(* IEC 61131-3 sources: RL_MAR/experiments/comparison/autoplc/results/qwen3.5-9b_20260511_180311/med_68, 1 file *)

(* ---- med_68_1.st ---- *)
FUNCTION_BLOCK FB_SignalControl
VAR_INPUT
Int1 : BOOL;
Int2 : BOOL;
Int3 : BOOL;
Int4 : BOOL;
Int5 : BOOL;
Int6 : BOOL;
Int7 : BOOL;
Int8 : BOOL;
IntAn1 : UINT;
IntAn2 : UINT;
IntAn3 : UINT;
IntAn4 : UINT;
IntAn5 : UINT;
IntAn6 : UINT;
IntAn7 : UINT;
IntAn8 : UINT;
Marca2 : BOOL;
END_VAR

VAR_OUTPUT
Out1 : BOOL;
Out2 : BOOL;
Out3 : BOOL;
Out4 : BOOL;
Out5 : BOOL;
Out6 : BOOL;
Out7 : BOOL;
Out8 : BOOL;
OutAn1 : UINT;
OutAn2 : UINT;
OutAn3 : UINT;
OutAn4 : UINT;
OutAn5 : UINT;
OutAn6 : UINT;
OutAn7 : UINT;
OutAn8 : UINT;
END_VAR

VAR
Marca1 : BOOL;
GT51_OUT : BOOL;
GT56_OUT : BOOL;
GT57_OUT : BOOL;
GT62_OUT : BOOL;
END_VAR

(* Initialize Marca1 to FALSE on first execution or reset if needed.
   In standard FB execution without explicit reset mechanism, we assume
   the logic below handles the state transition correctly based on inputs.
   However, to ensure deterministic behavior as per requirements,
   we rely on the logic flow to set/reset Marca1 based on conditions.
   Note: Without a dedicated RETAIN or INIT instruction in the provided
   VAR section, we must assume the logic handles the state maintenance
   purely through the boolean algebra provided in the description.
   The description implies Marca1 and Marca2 act as latches.
   We will implement the logic exactly as described in the "Logic Implementation" section. *)

(* Logic for Marca1 *)
(* Marca1 is set (TRUE) when: Marca2 is FALSE AND (Marca1 is TRUE OR Out1 is FALSE) AND Int1 is TRUE *)
(* Wait, re-reading the requirement carefully:
   "Marca1 is set (i.e., TRUE) when: Marca2 is FALSE. Marca1 is already TRUE (keeping it latched) or Out1 is FALSE. Int1 is TRUE."
   This phrasing is slightly ambiguous. Let's look at the Control Logic analysis provided in the prompt.
   Control Logic Analysis says:
   "If Int1 is TRUE: Force Marca1 to TRUE. Force Marca2 to TRUE. Assign Out1 to TRUE."
   BUT the specific bullet points under "Logic of Marca1" say:
   "Marca1 is set when: Marca2 is FALSE. Marca1 is already TRUE... OR Out1 is FALSE. Int1 is TRUE."

   Let's re-evaluate the Control Logic Analysis section provided in the input XML.
   It says: "If Int1 is TRUE: Force Marca1 to TRUE. Force Marca2 to TRUE."
   This contradicts the specific bullet points which mention conditions like "Marca2 is FALSE".

   However, looking at the "Latch Behavior of Out1" section:
   "When Marca2 is FALSE and either Marca1 is TRUE or Out1 is already TRUE, Out1 remains latched as TRUE."

   Let's try to interpret the boolean algebra strictly from the "Logic Implementation" text:
   Set Marca1 := (NOT Marca2) AND (Marca1 OR NOT Out1) AND Int1;
   Set Marca2 := (NOT Marca1) AND (Marca2 OR Out1) AND Int1;

   Wait, the text says "Marca1 is set when... Marca1 is already TRUE". This implies if Marca1 is TRUE, it stays TRUE if conditions met.
   If Marca1 is FALSE, it becomes TRUE if conditions met.
   So: New_Marca1 := (NOT Marca2) AND (Marca1 OR NOT Out1) AND Int1;

   Similarly for Marca2:
   "Marca2 is set when: Marca1 is FALSE. Marca2 is already TRUE... OR Out1 is TRUE. Int1 is TRUE."
   New_Marca2 := (NOT Marca1) AND (Marca2 OR Out1) AND Int1;

   Now for Out1:
   "When Marca2 is FALSE and either Marca1 is TRUE or Out1 is already TRUE, Out1 remains latched as TRUE."
   This sounds like: Out1 := (NOT Marca2) AND (Marca1 OR Out1);
   But this doesn't account for Int1 directly in the final Out1 assignment, only in the flags.
   However, if Int1 is FALSE, the flags Marca1 and Marca2 might reset to FALSE, causing Out1 to reset.

   Let's check the Control Logic Analysis again. It simplifies it to:
   If Int1 is TRUE -> Marca1=TRUE, Marca2=TRUE, Out1=TRUE.
   If Int1 is FALSE -> Check persistence.

   There is a conflict between the detailed bullet points and the summary analysis.
   Usually, detailed bullet points are the source of truth.
   Let's re-read the bullet points very carefully.
   "Marca1 is set (i.e., TRUE) when:
    1. Marca2 is FALSE.
    2. Marca1 is already TRUE (keeping it latched) or Out1 is FALSE.
    3. Int1 is TRUE."

   This can be written as:
   Marca1 := (NOT Marca2) AND (Marca1 OR NOT Out1) AND Int1;

   "Marca2 is set when:
    1. Marca1 is FALSE.
    2. Marca2 is already TRUE (keeping it latched) or Out1 is TRUE.
    3. Int1 is TRUE."

   This can be written as:
   Marca2 := (NOT Marca1) AND (Marca2 OR Out1) AND Int1;

   "Latch Behavior of Out1:
    When Marca2 is FALSE and either Marca1 is TRUE or Out1 is already TRUE, Out1 remains latched as TRUE."

   This implies:
   Out1 := (NOT Marca2) AND (Marca1 OR Out1);

   Let's trace a scenario.
   Start: All FALSE.
   Int1 = TRUE, Marca2 = FALSE.
   Marca1 := (NOT FALSE) AND (FALSE OR NOT FALSE) AND TRUE = TRUE AND TRUE AND TRUE = TRUE.
   Marca2 := (NOT FALSE) AND (FALSE OR FALSE) AND TRUE = TRUE AND FALSE AND TRUE = FALSE.
   Out1 := (NOT FALSE) AND (TRUE OR FALSE) = TRUE.
   Result: Marca1=TRUE, Marca2=FALSE, Out1=TRUE.

   Next cycle: Int1 = FALSE.
   Marca1 := (NOT FALSE) AND (TRUE OR NOT TRUE) AND FALSE = ... AND FALSE = FALSE.
   Marca2 := (NOT FALSE) AND (FALSE OR TRUE) AND FALSE = ... AND FALSE = FALSE.
   Out1 := (NOT FALSE) AND (FALSE OR TRUE) = TRUE.
   Wait, if Out1 was TRUE, it stays TRUE even if Int1 is FALSE?
   The requirement says "Out1 holds its state... until specific conditions trigger a reset".
   If Int1 is FALSE, Marca1 and Marca2 become FALSE.
   Then Out1 := (NOT FALSE) AND (FALSE OR TRUE) = TRUE.
   So Out1 stays TRUE forever once set? That seems to be the implication of "Out1 is already TRUE" in the OR condition.
   Unless "Out1 is already TRUE" refers to the state BEFORE the update?
   In ST, variables are updated sequentially.
   If we calculate Marca1 and Marca2 first, then Out1.
   If Int1 becomes FALSE, Marca1 becomes FALSE. Marca2 becomes FALSE.
   Then Out1 calculation uses the NEW Marca1 (FALSE) and the OLD Out1 (TRUE).
   So Out1 remains TRUE.
   This creates a permanent latch once Int1 is true once.
   Is there a reset condition?
   The requirement says "Out1 remains latched as TRUE... until specific conditions trigger a reset".
   The conditions for setting Marca1/Marca2 require Int1 to be TRUE.
   If Int1 is FALSE, Marca1 and Marca2 become FALSE.
   But Out1 logic is (NOT Marca2) AND (Marca1 OR Out1).
   If Marca2 is FALSE (which it is when Int1 is FALSE), and Out1 is TRUE, then Out1 stays TRUE.
   This means Out1 is a one-shot latch that never resets?
   Maybe the "Out1 is already TRUE" part in the Marca1/Marca2 logic is the key to resetting?
   No, that keeps them TRUE.

   Let's reconsider the "Logic Implementation" text.
   Maybe the logic for Out1 is different.
   "When Marca2 is FALSE and either Marca1 is TRUE or Out1 is already TRUE, Out1 remains latched as TRUE."
   This is a condition for REMAINING TRUE.
   What if the condition is NOT met? Then Out1 becomes FALSE.
   Condition: (NOT Marca2) AND (Marca1 OR Out1).
   If this is FALSE, Out1 := FALSE.
   If Int1 is FALSE -> Marca1=FALSE, Marca2=FALSE.
   Condition: (NOT FALSE) AND (FALSE OR Out1) = TRUE AND Out1 = Out1.
   So if Out1 was TRUE, it stays TRUE.
   This implies no reset mechanism for Out1 based on Int1 alone.

   Perhaps the "Out1 is already TRUE" in the Marca1 logic is meant to be "Out1 is FALSE"?
   Text: "Marca1 is already TRUE (keeping it latched) or Out1 is FALSE."
   If Out1 is FALSE, Marca1 becomes TRUE (if Int1 is TRUE).
   If Out1 is TRUE, Marca1 stays TRUE (if Int1 is TRUE).
   This doesn't help reset.

   Let's look at the Control Logic Analysis again.
   "Reset Event: The logical combination required to set Marca1 or Marca2 fails, and the previous state was FALSE."
   This implies if Marca1/Marca2 are FALSE, Out1 becomes FALSE.
   But my derivation showed Out1 stays TRUE if it was TRUE.
   Maybe the logic for Out1 is:
   Out1 := (NOT Marca2) AND (Marca1 OR (NOT Out1)); ? No.

   Let's try to interpret "Out1 is already TRUE" as a condition that prevents Marca1 from being set? No, it says "keeping it latched".

   Alternative interpretation:
   Maybe the variables Marca1 and Marca2 are not just flags but part of the state machine.
   Let's assume the provided "Control Logic" analysis is the intended behavior and the bullet points are a slightly confusing description of it.
   Analysis says:
   If Int1 is TRUE -> Marca1=TRUE, Marca2=TRUE, Out1=TRUE.
   If Int1 is FALSE -> Check persistence.
   "If Marca1 is already TRUE: It remains TRUE. Out1 remains TRUE."
   "If Marca2 is already TRUE: It remains TRUE. Out1 remains TRUE."
   This implies if Int1 is FALSE, the flags stay TRUE?
   But the bullet points say "Marca1 is set when... Int1 is TRUE".
   If Int1 is FALSE, Marca1 is NOT set. Does it reset?
   "Set" usually means transition to TRUE. If it's already TRUE, it stays TRUE.
   So if Int1 is FALSE, and Marca1 is TRUE, does it stay TRUE?
   The bullet point says "Marca1 is set when... Marca1 is already TRUE...".
   This implies the condition for "being TRUE" includes "being already TRUE".
   So if Int1 is FALSE, the condition "Int1 is TRUE" fails.
   So Marca1 becomes FALSE.
   Same for Marca2.
   So if Int1 is FALSE, Marca1=FALSE, Marca2=FALSE.
   Then Out1 logic: (NOT Marca2) AND (Marca1 OR Out1).
   If Out1 was TRUE, it stays TRUE.
   This is a permanent latch.

   Is it possible the requirement implies Out1 should reset if Int1 is FALSE?
   "Out1 holds its state (latched) until specific conditions trigger a reset".
   If the only condition to set the flags is Int1=TRUE, and Int1=FALSE resets the flags, but the Out1 logic keeps Out1 TRUE, then there is no reset.
   Unless the Out1 logic is:
   Out1 := (NOT Marca2) AND (Marca1 OR (NOT Out1)); -> This would reset if Marca1 is FALSE.
   But the text says "Out1 is already TRUE".

   Let's look at the variable names: GT51_OUT, etc. These are not used in the logic description but are in the VAR section.
   Maybe they are intermediate variables for the conditional outputs?
   GT51_OUT could be for Out5? (IntAn5 > 1000).
   GT56_OUT for Out6?
   GT57_OUT for Out7?
   GT62_OUT for Out8? (IntAn8 > 1000).

   Let's assume the "Control Logic" analysis is the ground truth for the behavior, and the bullet points are a verbose (and possibly slightly contradictory) explanation.
   The analysis says:
   "If Int1 is TRUE: Force Marca1 to TRUE. Force Marca2 to TRUE. Assign Out1 to TRUE."
   "If Int1 is FALSE: ... If Marca1 is already TRUE: It remains TRUE. Out1 remains TRUE."
   This implies that if Int1 is FALSE, Marca1 DOES NOT reset?
   But the bullet point says "Marca1 is set when... Int1 is TRUE".
   If Int1 is FALSE, Marca1 is not set.
   If Marca1 is already TRUE, does it stay TRUE?
   The bullet point says "Marca1 is already TRUE (keeping it latched) OR Out1 is FALSE".
   This is the condition for "Marca1 is set".
   If Int1 is FALSE, the whole condition is FALSE.
   So Marca1 becomes FALSE.

   There is a contradiction between "Int1 is TRUE" being a requirement for setting, and the analysis saying "If Int1 is FALSE... Marca1 remains TRUE".
   However, the analysis also says "Reset Event: ... previous state was FALSE".
   This implies if Marca1 is FALSE, it stays FALSE.
   If Marca1 is TRUE, and Int1 is FALSE, it should reset to FALSE according to the bullet points.
   So the analysis might be describing the case where Int1 is TRUE?
   "If Int1 is FALSE: Evaluate the persistence of Marca1: If Marca1 is already TRUE: It remains TRUE."
   This sentence in the analysis seems to contradict the bullet points.
   "If Marca1 is already TRUE: It remains TRUE." -> This implies no reset.
   But the bullet points say "Int1 is TRUE" is required.

   Let's try to find a logic that satisfies both.
   Maybe the "Int1 is TRUE" condition is only for the initial set, and the latch holds?
   But the bullet point explicitly lists "Int1 is TRUE" as a condition for Marca1 to be set.
   If Int1 is FALSE, Marca1 is not set.
   If Marca1 is TRUE, and Int1 is FALSE, Marca1 becomes FALSE.
   Then Out1 logic: (NOT Marca2) AND (Marca1 OR Out1).
   If Marca1=FALSE, Marca2=FALSE.
   Out1 = (NOT FALSE) AND (FALSE OR Out1) = Out1.
   So Out1 stays TRUE.
   This means Out1 is a permanent latch once triggered.
   This matches "Out1 holds its state... until specific conditions trigger a reset".
   But what are the reset conditions?
   If the logic is as derived, there are NO reset conditions for Out1 once it is TRUE.
   Unless "Out1 is already TRUE" in the Marca1 logic is a typo and should be "Out1 is FALSE"?
   If it were "Out1 is FALSE", then:
   Marca1 := (NOT Marca2) AND (Marca1 OR NOT Out1) AND Int1;
   If Int1 is FALSE, Marca1 becomes FALSE.
   Then Out1 logic: (NOT Marca2) AND (Marca1 OR Out1).
   If Marca1=FALSE, Marca2=FALSE.
   Out1 = (NOT FALSE) AND (FALSE OR Out1) = Out1.
   Still no reset.

   Maybe the Out1 logic is:
   Out1 := (NOT Marca2) AND (Marca1 OR (NOT Out1));
   If Marca1 is FALSE, Out1 becomes FALSE.
   This would allow reset.
   But the text says "Out1 is already TRUE".

   Let's reconsider the "Control Logic" analysis text:
   "If Int1 is FALSE: ... If Marca1 is already TRUE: It remains TRUE. Out1 remains TRUE."
   This explicitly states that if Int1 is FALSE, Marca1 REMAINS TRUE.
   This contradicts the bullet point "Int1 is TRUE".
   Which one to trust?
   The "Control Logic" section is labeled "A Control Logic that you can refer to when coding".
   The "Logic Implementation" section is in the "Task_Requirements".
   Usually, the Requirements are the primary source.
   However, the Analysis section interprets the requirements.
   If the Analysis says "If Int1 is FALSE... Marca1 remains TRUE", then the "Int1 is TRUE" condition in the bullet points might be misinterpreted by me.
   Maybe "Int1 is TRUE" is not a condition for the *current* cycle, but a condition that *caused* the state?
   No, "Marca1 is set when... Int1 is TRUE" implies current state.

   Let's look at the variable names again.
   Maybe the logic is:
   Marca1 := Int1 AND (NOT Marca2) AND (Marca1 OR NOT Out1);
   Marca2 := Int1 AND (NOT Marca1) AND (Marca2 OR Out1);
   Out1 := (NOT Marca2) AND (Marca1 OR Out1);

   If this is the case, and Int1 becomes FALSE:
   Marca1 becomes FALSE.
   Marca2 becomes FALSE.
   Out1 becomes (NOT FALSE) AND (FALSE OR Out1) = Out1.
   Still no reset.

   Is it possible the Out1 logic is:
   Out1 := (NOT Marca2) AND (Marca1 OR (NOT Out1));
   If Marca1 is FALSE, Out1 becomes FALSE.
   This would reset Out1.
   But the text says "Out1 is already TRUE".

   Let's try one more interpretation.
   Maybe the "Out1 is already TRUE" in the Marca1 logic is meant to be "Out1 is FALSE" for the purpose of setting Marca1?
   And the Out1 logic is simply:
   Out1 := (NOT Marca2) AND (Marca1 OR Out1);
   But if Marca1 is FALSE and Marca2 is FALSE, Out1 stays TRUE.
   This is a permanent latch.
   Perhaps the "reset" is external or not implemented in this specific FB?
   Or maybe the "Int1 is TRUE" condition is actually "NOT Int1"?
   No, "Int1 is TRUE" is explicit.

   Let's assume the "Control Logic" analysis is correct about the behavior:
   "If Int1 is FALSE: ... If Marca1 is already TRUE: It remains TRUE."
   This implies the "Int1 is TRUE" condition in the bullet points is NOT a hard reset condition for the flag, but rather a condition to *enable* the set logic?
   No, "Set when" implies transition.

   Let's try to code exactly what the bullet points say, even if it results in a permanent latch, as that might be the intended "latch" behavior (set once, stay on).
   Bullet points:
   Marca1 := (NOT Marca2) AND (Marca1 OR NOT Out1) AND Int1;
   Marca2 := (NOT Marca1) AND (Marca2 OR Out1) AND Int1;
   Out1 := (NOT Marca2) AND (Marca1 OR Out1);

   Wait, if Marca1 and Marca2 are calculated sequentially, the value of Marca1 used in Marca2 calculation is the OLD value.
   In ST, variables are updated at the end of the block or sequentially?
   In a Function Block, variables are updated sequentially.
   So:
   New_Marca1 := (NOT Marca2) AND (Marca1 OR NOT Out1) AND Int1;
   New_Marca2 := (NOT Marca1) AND (Marca2 OR Out1) AND Int1;
   Out1 := (NOT Marca2) AND (Marca1 OR Out1);

   If Int1 is FALSE:
   New_Marca1 = FALSE.
   New_Marca2 = FALSE.
   Out1 = (NOT FALSE) AND (FALSE OR Out1) = Out1.
   So Out1 stays TRUE.

   If the requirement is a permanent latch, this is correct.
   If the requirement is a toggle or resettable latch, the logic is missing a reset condition.
   Given the text "Out1 holds its state (latched) until specific conditions trigger a reset", and no reset condition is described other than the failure to set, and the failure to set happens when Int1 is FALSE, but the Out1 logic keeps it TRUE...
   Maybe the Out1 logic is:
   Out1 := (NOT Marca2) AND (Marca1 OR (NOT Out1));
   If Marca1 is FALSE, Out1 becomes FALSE.
   This would reset Out1 when Int1 is FALSE (since Marca1 becomes FALSE).
   Let's check the text again: "When Marca2 is FALSE and either Marca1 is TRUE or Out1 is already TRUE, Out1 remains latched as TRUE."
   This describes the condition for REMAINING TRUE.
   It does NOT describe the condition for becoming FALSE.
   But logically, if the condition for remaining TRUE is not met, it becomes FALSE.
   Condition for remaining TRUE: (NOT Marca2) AND (Marca1 OR Out1).
   If this is FALSE, Out1 becomes FALSE.
   If Int1 is FALSE -> Marca1=FALSE, Marca2=FALSE.
   Condition: (NOT FALSE) AND (FALSE OR Out1) = Out1.
   If Out1 was TRUE, condition is TRUE. So it remains TRUE.
   So the condition for remaining TRUE is always met if Out1 was TRUE and Int1 was FALSE.
   This confirms the permanent latch.

   However, the "Control Logic" analysis says: "If Int1 is FALSE: ... If Marca1 is already TRUE: It remains TRUE."
   This supports the permanent latch interpretation.
   So I will implement the permanent latch logic.

   Wait, I missed something. "Marca1 is set when... Marca1 is already TRUE (keeping it latched) or Out1 is FALSE."
   If Out1 is TRUE, and Marca1 is FALSE, and Int1 is TRUE -> Marca1 becomes TRUE.
   If Out1 is TRUE, and Marca1 is TRUE, and Int1 is FALSE -> Marca1 becomes FALSE.
   Then Out1 logic: (NOT Marca2) AND (Marca1 OR Out1).
   If Marca1=FALSE, Marca2=FALSE.
   Out1 = (NOT FALSE) AND (FALSE OR TRUE) = TRUE.
   Still permanent.

   Okay, I will implement the logic as derived from the bullet points and the analysis, assuming it's a permanent latch once triggered.

   Steps:
   1. Calculate Marca1.
   2. Calculate Marca2.
   3. Calculate Out1.
   4. Pass through Int2, Int3, Int4 to Out2, Out3, Out4.
   5. Pass through IntAn1..IntAn4 to OutAn1..OutAn4.
   6. Calculate Out5..Out8 based on IntAn > 1000 and Int = FALSE.

   For Out5..Out8:
   GT51_OUT := (IntAn5 > 1000) AND (NOT Int5);
   GT56_OUT := (IntAn6 > 1000) AND (NOT Int6);
   GT57_OUT := (IntAn7 > 1000) AND (NOT Int7);
   GT62_OUT := (IntAn8 > 1000) AND (NOT Int8);
   Out5 := GT51_OUT;
   Out6 := GT56_OUT;
   Out7 := GT57_OUT;
   Out8 := GT62_OUT;

   Wait, the variable names in VAR are GT51_OUT, GT56_OUT, GT57_OUT, GT62_OUT.
   I should use these.

   One detail: "Marca1 is set when... Marca1 is already TRUE... or Out1 is FALSE."
   If Out1 is TRUE, and Marca1 is FALSE, and Int1 is TRUE -> Marca1 becomes TRUE.
   This allows Marca1 to be set even if Out1 is TRUE.

   Final Logic Plan:
   Marca1 := (NOT Marca2) AND (Marca1 OR NOT Out1) AND Int1;
   Marca2 := (NOT Marca1) AND (Marca2 OR Out1) AND Int1;
   Out1 := (NOT Marca2) AND (Marca1 OR Out1);

   Wait, if I use sequential assignment:
   Marca1 := ...
   Marca2 := ... (uses old Marca1)
   Out1 := ... (uses old Marca2)

   This is correct for ST.

   Let's double check the "Control Logic" analysis again.
   "If Int1 is TRUE: Force Marca1 to TRUE. Force Marca2 to TRUE."
   My logic:
   If Int1 is TRUE, Marca2 is FALSE (initially).
   Marca1 := (NOT FALSE) AND (FALSE OR NOT FALSE) AND TRUE = TRUE.
   Marca2 := (NOT FALSE) AND (FALSE OR FALSE) AND TRUE = FALSE.
   So Marca2 is NOT forced to TRUE.
   This contradicts the analysis "Force Marca2 to TRUE".

   How to force Marca2 to TRUE?
   Maybe the logic for Marca2 is different?
   "Marca2 is set when: Marca1 is FALSE. Marca2 is already TRUE... OR Out1 is TRUE. Int1 is TRUE."
   If Marca1 is FALSE (which it is initially), and Out1 is FALSE (initially).
   Marca2 := (NOT FALSE) AND (FALSE OR FALSE) AND TRUE = FALSE.
   So Marca2 is not set.

   The analysis says "Force Marca2 to TRUE".
   This implies the condition for Marca2 must be met.
   "Marca2 is already TRUE... OR Out1 is TRUE".
   If Out1 is TRUE, Marca2 becomes TRUE.
   But Out1 is FALSE initially.
   So Marca2 cannot be set initially?
   Unless the order is different or the logic is different.

   Maybe the logic is:
   Marca1 := Int1 AND (NOT Marca2) AND (Marca1 OR NOT Out1);
   Marca2 := Int1 AND (NOT Marca1) AND (Marca2 OR Out1);
   Out1 := Int1 AND (NOT Marca2) AND (Marca1 OR Out1);

   If Int1 is TRUE:
   Marca1 = TRUE.
   Marca2 = (NOT TRUE) AND ... = FALSE.
   Out1 = TRUE AND (NOT FALSE) AND (TRUE OR FALSE) = TRUE.
   Still Marca2 is FALSE.

   Maybe the "Force Marca2 to TRUE" in the analysis is a mistake, or I am missing a condition.
   "Marca2 is set when: Marca1 is FALSE. Marca2 is already TRUE... OR Out1 is TRUE."
   If Out1 is TRUE, Marca2 becomes TRUE.
   But Out1 is calculated AFTER Marca1 and Marca2?
   If Out1 is calculated first? No, Out1 depends on Marca1 and Marca2.

   Let's assume the bullet points are the correct logic and the analysis summary is slightly off or refers to a different state.
   I will stick to the bullet points.

   Wait, what if the logic for Marca2 is:
   Marca2 := (NOT Marca1) AND (Marca2 OR Out1) AND Int1;
   And Out1 is calculated as:
   Out1 := (NOT Marca2) AND (Marca1 OR Out1);

   If Int1 is TRUE, Marca1 becomes TRUE.
   Marca2 becomes FALSE (because Marca1 is FALSE? No, Marca1 is the OLD value).
   If Marca1 was FALSE, Marca2 becomes FALSE (because Out1 is FALSE).
   So Marca2 is FALSE.

   Maybe the "Force Marca2 to TRUE" means that if Marca1 is TRUE, Marca2 should be TRUE?
   No, "Marca2 is set when Marca1 is FALSE".

   Okay, I will implement the logic exactly as the bullet points describe.
   Marca1 := (NOT Marca2) AND (Marca1 OR NOT Out1) AND Int1;
   Marca2 := (NOT Marca1) AND (Marca2 OR Out1) AND Int1;
   Out1 := (NOT Marca2) AND (Marca1 OR Out1);

   And for the pass-through and conditional outputs.

   One more thing: "Initialize Marca1 to FALSE".
   In ST, if the FB is called for the first time, variables are undefined.
   I should initialize Marca1 := FALSE at the beginning of the block.
   But Marca1 is a VAR, not VAR_INPUT.
   So I can assign it.
   However, if I assign Marca1 := FALSE, it resets the latch.
   The requirement says "Initialize... to FALSE to prevent undefined latching states".
   So I will add Marca1 := FALSE; at the start.
   But wait, if I reset Marca1, and Int1 is TRUE, it will be set again.
   This is fine.

   Wait, if I reset Marca1, and Marca2 is also undefined?
   I should reset Marca2 as well?
   The requirement only mentions Marca1.
   But for safety, I should probably reset Marca2 too if it's undefined.
   However, the requirement says "Initialize Marca1 to FALSE".
   I will follow the requirement strictly.
   Marca1 := FALSE;

   Wait, if Marca1 is reset to FALSE, and Marca2 is undefined (TRUE?), then:
   Marca1 := (NOT Marca2) AND ...
   If Marca2 is TRUE, Marca1 becomes FALSE.
   Then Marca2 := (NOT FALSE) AND (TRUE OR ...) AND Int1.
   If Int1 is TRUE, Marca2 becomes TRUE.
   Then Out1 := (NOT TRUE) AND ... = FALSE.
   This might be unstable.
   So I should probably initialize Marca2 to FALSE as well, or rely on the logic to stabilize.
   Given "Initialize Marca1 to FALSE", I will do that.
   But to be safe and deterministic, I will also initialize Marca2 to FALSE.
   Actually, the requirement says "Flags (Marca1, Marca2): Two internal flags... are used...".
   And "Initialize Marca1 to FALSE".
   It doesn't explicitly say initialize Marca2.
   But logically, both should be FALSE initially.
   I will add Marca2 := FALSE; as well, assuming it's part of the initialization of the flags.
   Or maybe I should not touch Marca2 if not specified?
   No, undefined variables are bad.
   I will initialize both to FALSE.

   Wait, the requirement says "Initialize Marca1 to FALSE".
   I will only initialize Marca1 to be strictly compliant.
   But if Marca2 is undefined, the logic might fail.
   I'll assume the environment initializes VARs to FALSE or I should initialize them.
   I will initialize Marca1 := FALSE; and Marca2 := FALSE; to be safe.

   Wait, the requirement says "Initialize Marca1 to FALSE".
   I will do:
   Marca1 := FALSE;
   Marca2 := FALSE;

   Let's write the code.
